SYSTEM TESTPAR_SYS (* Test Setting of Parameters in a System Configuration *)
  (* Standard: 61499-1 *)
  (* Version 0.0, 2004-12-16, JHC, Rockwell Automation *)
  DEVICE HMI : FRAME_DEVICE(BOUNDS := [100,100,75,50])
    RESOURCE RES1 : PANEL_RESOURCE
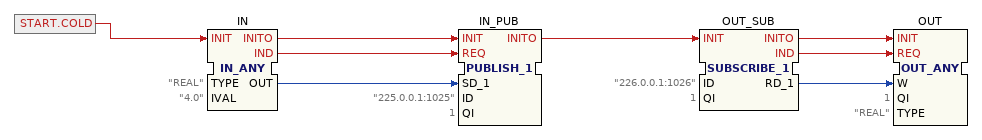
      FBS
        IN : IN_ANY(TYPE := "REAL", IVAL := "4.0");
        IN_PUB : PUBLISH_1(ID := "225.0.0.1:1025", QI := 1);
        OUT_SUB : SUBSCRIBE_1(ID := "226.0.0.1:1026", QI := 1);
        OUT : OUT_ANY(QI := 1, TYPE := "REAL");
      END_FBS
      EVENT_CONNECTIONS
        START.COLD TO IN.INIT;
        IN.INITO TO IN_PUB.INIT;
        IN.IND TO IN_PUB.REQ;
        IN_PUB.INITO TO OUT_SUB.INIT;
        OUT_SUB.INITO TO OUT.INIT;
        OUT_SUB.IND TO OUT.REQ;
      END_CONNECTIONS
      DATA_CONNECTIONS
        IN.OUT TO IN_PUB.SD_1;
        OUT_SUB.RD_1 TO OUT.W;
      END_CONNECTIONS
    END_RESOURCE
  END_DEVICE
  DEVICE TEST : TESTPAR_DEV
  END_DEVICE
END_SYSTEM
